(* CODESYS project my-demo.ecp

Project tree, tasks and I/O mapping:
  GenericDummyMasterDevice : Generic Master, WAGO, order no. None, version 1.0.0.0
  PFC200_CS_2ETH_RS : 750-8202 PFC200 2ETH RS, WAGO, order no. 0750-8202, version 1.4.1.22
    application Application
      libraries: 
      task PLC_Task (cyclic, interval t#10ms, priority 14) calls PLC_PRG
      program PLC_PRG [ST]
    DeviceAdapter
    Kbus : Kbus, WAGO, version 1.3.0.0
        unmapped channels: K-BUS diagnostics
      _8_DO_DI_Generic : 075x-8DO8DI, WAGO, order no. 075x-8DO8DI, version 0.0.0.11
          settings: K-BUS Module slot index = 1
          input  Application.PLC_PRG.button : BOOL  // _IN._IN
          output Application.PLC_PRG.led : BOOL  // _OUT._OUT
          unmapped channels: _IN, _OUT
        DeviceAdapter
    MODBUS
      MODBUS : MODBUS, WAGO, order no. n/a, version 1.1.1.13
    Serial
      COM1 : COM1, WAGO, version 0.0.0.19
*)

// PFC200_CS_2ETH_RS/Application/PLC_PRG
PROGRAM PLC_PRG
VAR
	counter: INT := 0;
	led: BOOL := FALSE;
	button: BOOL := TRUE;
END_VAR

IF (button) THEN
	counter := counter + 1;
	IF (counter = 50) THEN
		counter := 0;
		led := NOT led;
	END_IF
ELSE
	led := FALSE;
END_IF

END_PROGRAM
